FUNCTION_BLOCK FB_StrategyTravelByBycicle IMPLEMENTS I_Strategy
VAR_INPUT
END_VAR
VAR_OUTPUT
END_VAR
VAR
END_VAR

METHOD execute
VAR_INPUT
	in_rDistance		:REAL;
END_VAR
ADSLOGSTR(msgCtrlMask:= ADSLOG_MSGTYPE_ERROR, msgFmtStr:= 'Travel time by bycicle: %s min', strArg:= TO_STRING(in_rDistance * 4.0));
END_METHOD

END_FUNCTION_BLOCK

(* stored: Version 1.1.0.1
   POU FB_StrategyTravelByBycicle: Id {448a735d-bb15-44df-8798-4980087a678a}, SpecialFunc None
   Method execute: Id {7f87578f-4a3c-4ac0-8f7c-41a21a3370ad} *)
